Staubli VAL3: onStop.pgx

public program onStop(string& x_sItem[])
  local num l_nResult
begin
  // reload all the template
  l_nResult=extCall0:libLoad("Disk://..//templates/call")
  delay(0)
  l_nResult=l_nResult+extCall1:libLoad("Disk://..//templates/call")
  delay(0)
  l_nResult=l_nResult+extCall2:libLoad("Disk://..//templates/call")
  delay(0)
  l_nResult=l_nResult+extCall3:libLoad("Disk://..//templates/call")
  delay(0)
  l_nResult=l_nResult+extCall4:libLoad("Disk://..//templates/call")
  delay(0)
  l_nResult=l_nResult+extCall5:libLoad("Disk://..//templates/call")
  delay(0)
  l_nResult=l_nResult+extCall6:libLoad("Disk://..//templates/call")
  delay(0)
  l_nResult=l_nResult+extCall7:libLoad("Disk://..//templates/call")
  delay(0)
  l_nResult=l_nResult+extCall8:libLoad("Disk://..//templates/call")
  delay(0)
  l_nResult=l_nResult+extCall9:libLoad("Disk://..//templates/call")
  delay(0)
  l_nResult=l_nResult+extCall10:libLoad("Disk://..//templates/call")
  delay(0)
  l_nResult=l_nResult+extCall11:libLoad("Disk://..//templates/call")
  delay(0)
  l_nResult=l_nResult+extCall12:libLoad("Disk://..//templates/call")
  delay(0)
  l_nResult=l_nResult+extCall13:libLoad("Disk://..//templates/call")
  delay(0)
  l_nResult=l_nResult+extCall14:libLoad("Disk://..//templates/call")
  delay(0)
  l_nResult=l_nResult+extCall15:libLoad("Disk://..//templates/call")
  delay(0)
  l_nResult=l_nResult+extCall16:libLoad("Disk://..//templates/call")
  delay(0)
  l_nResult=l_nResult+extCall17:libLoad("Disk://..//templates/call")
  delay(0)
  l_nResult=l_nResult+extCall18:libLoad("Disk://..//templates/call")
  delay(0)
  l_nResult=l_nResult+extCall19:libLoad("Disk://..//templates/call")
  delay(0)
end
